FUNCTION_BLOCK FB_SetAndActivateConfig
VAR_IN_OUT
 stPiezoStage  : ST_PiezoStage;
END_VAR

VAR_INPUT
     bExecute  : BOOL := FALSE;
     nIndex     : WORD ; 		   (* CoE Object Index *)
     nSubIndex  : BYTE ; 			   (* Subindex of CoE Object *)
     nValue		: DINT;
END_VAR

VAR_OUTPUT
     bBusy   : BOOL := FALSE;
     bDone   : BOOL := FALSE;
     bError  : BOOL := FALSE;
     nErrorId  : UDINT := 0;
END_VAR
VAR
 fbSdoWrite : FB_EcCoESdoWrite;
END_VAR

IF NOT fbSdoWrite.bBusy THEN
    bExecute := FALSE;
    IF NOT fbSdoWrite.bError THEN
        (* write successful *)
        bError := FALSE;
        nErrorId := 0;
    ELSE
        (* write failed *)
        bError := fbSdoWrite.bError;
        nErrorId := fbSdoWrite.nErrId;

    END_IF

    fbSdoWrite(bExecute := FALSE);
END_IF

END_FUNCTION_BLOCK

(* stored: Version 1.1.0.1
   POU FB_SetAndActivateConfig: Id {8d5a249c-2e29-458b-823b-6fdba433baa6}, SpecialFunc None *)
